	fb103StartQuiescentMode.ipDALICommunication := ipDALICommunication;
	fb103StopQuiescentMode.ipDALICommunication := ipDALICommunication;
	fb253QueryShortCircuit.ipDALICommunication := ipDALICommunication;
	fb253QueryOpenCircuit.ipDALICommunication := ipDALICommunication;
	fb207QueryLoadDecrease.ipDALICommunication := ipDALICommunication;
	fb207QueryLoadIncrease.ipDALICommunication := ipDALICommunication;
	fb253QueryThermalShutDown.ipDALICommunication := ipDALICommunication;
	fb207QueryThermalOverload.ipDALICommunication := ipDALICommunication;
	fb207QueryReferenceMeasurementFailed.ipDALICommunication := ipDALICommunication;
	fb207QueryDimmingCurve.ipDALICommunication := ipDALICommunication;
	fb207QueryFastFadeTime.ipDALICommunication := ipDALICommunication;
	fb102QueryExtendedVersionNumber.ipDALICommunication := ipDALICommunication;
	fb207ReferenceSystemPower.ipDALICommunication := ipDALICommunication;
	fb207SelectDimmingCurve.ipDALICommunication := ipDALICommunication;
	fb207SetFastFadeTime.ipDALICommunication := ipDALICommunication;
	fb207QueryFeatures.ipDALICommunication := ipDALICommunication;
	fb207QueryControlGearType.ipDALICommunication := ipDALICommunication;
{endregion}
{region "Read Status}
5:
{region "Start Qiescent Mode"}
	fb103StartQuiescentMode(bStart := TRUE,
							eAddressType := Tc3_DALI.E_DALIAddressType.Broadcast,
							eCommandPriority := Tc3_DALI.E_DALICommandPriority.Middle);
	IF (NOT fb103StartQuiescentMode.bBusy) THEN
		fb103StartQuiescentMode(bStart:= FALSE);
		nStep := 10;
	END_IF
{endregion}
10:
{region "Query Short Circuit"}
	fb253QueryShortCircuit(	bStart := TRUE,
							nAddress := nAddress,
							eAddressType := Tc3_DALI.E_DALIAddressType.Short,
							eCommandPriority := Tc3_DALI.E_DALICommandPriority.Middle);
	IF (NOT fb253QueryShortCircuit.bBusy) THEN
		fb253QueryShortCircuit(bStart := FALSE);
		sShortCircuit := SEL(fb253QueryShortCircuit.bLightSourceShortCircuit, 'No', 'Yes');
		nStep := 20;
	END_IF
{endregion}
20:
{region "Query Open Circuit"}
	fb253QueryOpenCircuit(	bStart := TRUE,
							nAddress := nAddress,
							eAddressType := Tc3_DALI.E_DALIAddressType.Short,
							eCommandPriority := Tc3_DALI.E_DALICommandPriority.Middle);
	IF (NOT fb253QueryOpenCircuit.bBusy) THEN
		fb253QueryOpenCircuit(bStart := FALSE);
		sOpenCircuit := SEL(fb253QueryOpenCircuit.bLightSourceOpenCircuit, 'No', 'Yes');
		nStep := 30;
	END_IF
{endregion}
30:
{region "Query Load Decrease"}
	fb207QueryLoadDecrease(	bStart := TRUE,
							nAddress := nAddress,
							eAddressType := Tc3_DALI.E_DALIAddressType.Short,
							eCommandPriority := Tc3_DALI.E_DALICommandPriority.Middle);
	IF (NOT fb207QueryLoadDecrease.bBusy) THEN
		fb207QueryLoadDecrease(bStart := FALSE);
		sLoadDecrease := SEL(fb207QueryLoadDecrease.bLoadDecrease, 'No', 'Yes');
		nStep := 40;
	END_IF
{endregion}
40:
{region "Query Load Increase"}
	fb207QueryLoadIncrease(	bStart := TRUE,
							nAddress := nAddress,
							eAddressType := Tc3_DALI.E_DALIAddressType.Short,
							eCommandPriority := Tc3_DALI.E_DALICommandPriority.Middle);
	IF (NOT fb207QueryLoadIncrease.bBusy) THEN
		fb207QueryLoadIncrease(bStart := FALSE);
		sLoadIncrease := SEL(fb207QueryLoadIncrease.bLoadIncrease, 'No', 'Yes');
		nStep := 80;
	END_IF
{endregion}
80:
{region "Query Thermal Shut Down"}
	fb253QueryThermalShutDown(	bStart := TRUE,
								nAddress := nAddress,
								eAddressType := Tc3_DALI.E_DALIAddressType.Short,
								eCommandPriority := Tc3_DALI.E_DALICommandPriority.Middle);
	IF (NOT fb253QueryThermalShutDown.bBusy) THEN
		fb253QueryThermalShutDown(bStart := FALSE);
		sThermalShutDown := SEL(fb253QueryThermalShutDown.bLightSourceThermalShutdown, 'No', 'Yes');
		nStep := 90;
	END_IF
{endregion}
90:
{region "Query Thermal Overload"}
	fb207QueryThermalOverload(	bStart := TRUE,
								nAddress := nAddress,
								eAddressType := Tc3_DALI.E_DALIAddressType.Short,
								eCommandPriority := Tc3_DALI.E_DALICommandPriority.Middle);
	IF (NOT fb207QueryThermalOverload.bBusy) THEN
		fb207QueryThermalOverload(bStart := FALSE);
		sThermalOverload := SEL(fb207QueryThermalOverload.bThermalOverload, 'No', 'Yes');
		nStep := 100;
	END_IF
{endregion}
100:
{region "Query Reference Measurement Failed"}
	fb207QueryReferenceMeasurementFailed(	bStart := TRUE,
											nAddress := nAddress,
											eAddressType := Tc3_DALI.E_DALIAddressType.Short,
											eCommandPriority := Tc3_DALI.E_DALICommandPriority.Middle);
	IF (NOT fb207QueryReferenceMeasurementFailed.bBusy) THEN
		fb207QueryReferenceMeasurementFailed(bStart := FALSE);
		sReferenceMeasurementFailed := SEL(fb207QueryReferenceMeasurementFailed.bReferenceMeasurementFailed, 'No', 'Yes');
		nStep := 110;
	END_IF
{endregion}
110:
{region "Query Dimming Curve"}
	fb207QueryDimmingCurve(	bStart := TRUE,
							nAddress := nAddress,
							eAddressType := Tc3_DALI.E_DALIAddressType.Short,
							eCommandPriority := Tc3_DALI.E_DALICommandPriority.Middle,
							eDimmingCurve => eDimmingCurve);
	IF (NOT fb207QueryDimmingCurve.bBusy) THEN
		fb207QueryDimmingCurve(bStart := FALSE);
		nStep := 120;
	END_IF
{endregion}
120:
{region "Query Fast Fade Time"}
	fb207QueryFastFadeTime(	bStart := TRUE,
							nAddress := nAddress,
							eAddressType := Tc3_DALI.E_DALIAddressType.Short,
							eCommandPriority := Tc3_DALI.E_DALICommandPriority.Middle,
							eFastFadeTime => eFastFadeTime);
	IF (NOT fb207QueryFastFadeTime.bBusy) THEN
		fb207QueryFastFadeTime(bStart := FALSE);
		nStep := 130;
	END_IF
{endregion}
130:
{region "Query Extended Version Number"}
	fb102QueryExtendedVersionNumber(bStart := TRUE,
									nAddress := nAddress,
									eAddressType := Tc3_DALI.E_DALIAddressType.Short,
									eCommandPriority := Tc3_DALI.E_DALICommandPriority.Middle,
									eDeviceType := E_DALIDeviceType.DT06LEDModule,
									nExtendedVersionNumber => nExtendedVersionNumber);
	IF (NOT fb102QueryExtendedVersionNumber.bBusy) THEN
		fb102QueryExtendedVersionNumber(bStart := FALSE);
		nStep := 135;
	END_IF
{endregion}
135:
{region "Stop Qiescent Mode"}
	fb103StopQuiescentMode(	bStart := TRUE,
							eAddressType := Tc3_DALI.E_DALIAddressType.Broadcast,
							eCommandPriority := Tc3_DALI.E_DALICommandPriority.Middle);
	IF (NOT fb103StopQuiescentMode.bBusy) THEN
		fb103StopQuiescentMode(	bStart := FALSE);
		nStep := 0;
	END_IF
{endregion}
{endregion}

{region "Read Parameter"}
200:
{region "Start Qiescent Mode"}
	fb103StartQuiescentMode(bStart := TRUE,
							eAddressType := Tc3_DALI.E_DALIAddressType.Broadcast,
							eCommandPriority := Tc3_DALI.E_DALICommandPriority.Middle);
	IF (NOT fb103StartQuiescentMode.bBusy) THEN
		fb103StartQuiescentMode(bStart:= FALSE);
		nStep := 210;
	END_IF
{endregion}
210:
{region "Query Features"}
	fb207QueryFeatures(	bStart := TRUE,
						nAddress := nAddress,
						eAddressType := Tc3_DALI.E_DALIAddressType.Short,
						eCommandPriority := Tc3_DALI.E_DALICommandPriority.Middle,
						nFeatures => nFeatures);

	IF (NOT fb207QueryFeatures.bBusy) THEN
		fb207QueryFeatures(bStart := FALSE);
		bQueryShortCircuitEnabled := nFeatures.0;
		bQueryIdleTimeDetectionEnabled := nFeatures.1;
		bQueryLoadDecreaseEnabled := nFeatures.2;
		bQueryLoadIncreaseEnabled := nFeatures.3;
		bQueryCurrentProtectionDevicePresent := nFeatures.4;
		bQueryThermalSwitchEnabled := nFeatures.5;
		bQueryReductionOfLuminouFluxRegardingThermalOverloadEnabled := nFeatures.6;
		bPhysicalSelectionSupported := nFeatures.7;
		nStep := 215;
	END_IF
{endregion}
215:
{region "Query control Gear Type"}
	fb207QueryControlGearType(	bStart := TRUE, 
								nAddress := nAddress,
								eAddressType := Tc3_DALI.E_DALIAddressType.Short,
								eCommandPriority := Tc3_DALI.E_DALICommandPriority.Middle,
								nControlGearType => nControlGearType);
	IF (NOT fb207QueryControlGearType.bBusy) THEN
		fb207QueryControlGearType(bStart := FALSE);
		bLEDModule	:= nControlGearType.1;
		nStep := 220;
	END_IF
{endregion}
220:
{region "Stop Qiescent Mode"}
	fb103StopQuiescentMode(	bStart := TRUE,
							eAddressType := Tc3_DALI.E_DALIAddressType.Broadcast,
							eCommandPriority := Tc3_DALI.E_DALICommandPriority.Middle);
	IF (NOT fb103StopQuiescentMode.bBusy) THEN
		fb103StopQuiescentMode(	bStart := FALSE);
		nStep := 0;
	END_IF
{endregion}
{endregion}

{region "Write"}
1000:
{region "Reference System Power"}
	fb207ReferenceSystemPower(	bStart := TRUE,
								nAddress := nAddress,
								eAddressType := Tc3_DALI.E_DALIAddressType.Short,
								eCommandPriority := Tc3_DALI.E_DALICommandPriority.Middle);
	IF (NOT fb207ReferenceSystemPower.bBusy) THEN
		fb207ReferenceSystemPower(bStart := FALSE);
		nStep := 0;
	END_IF
{endregion}
1030:
{region "Select Dimming Curve"}
	fb207SelectDimmingCurve(bStart := TRUE,
							nAddress := nAddress,
							eAddressType := Tc3_DALI.E_DALIAddressType.Short,
							eCommandPriority := Tc3_DALI.E_DALICommandPriority.Middle,
							eDimmingCurve := eDimmingCurve);
	IF (NOT fb207SelectDimmingCurve.bBusy) THEN
		fb207SelectDimmingCurve(bStart := FALSE);
		nStep := 1040;
	END_IF
{endregion}
1040:
{region "Set Fast Fade Time"}
	fb207SetFastFadeTime(bStart := TRUE,
						nAddress := nAddress,
						eAddressType := Tc3_DALI.E_DALIAddressType.Short,
						eCommandPriority := Tc3_DALI.E_DALICommandPriority.Middle,
						eFastFadeTime := eFastFadeTime);
	IF (NOT fb207SetFastFadeTime.bBusy) THEN
		fb207SetFastFadeTime(bStart := FALSE);
		nStep := 0;
	END_IF
{endregion}
{endregion}
END_CASE

END_FUNCTION_BLOCK

// ---- POUs/EnOcean/P_EnOcean.TcPOU
PROGRAM P_EnOcean
VAR
	fbKL6581			: FB_KL6581;
	stKL6581_in  AT %I* : KL6581_INPUT;
	stKL6581_out AT %Q*	: KL6581_OUTPUT;
	stKL6581			: STR_KL6581;
	bInitCom			: BOOL := TRUE;
	
	arrEnOcean_Search	: ARRAY [1..8] OF FB_EnOcean_Search;
	nSearchIdx			: BYTE;
	bSerach				: BOOL;
	arrDevices			: ARRAY [1..8] OF INT;
	arrID					: ARRAY [1..8, 0..255] OF DWORD;

	//Trykknapper på gange
	fbGang_1_216_Tryk_Pendler    							: FB_Rec_RPS_Switch;	
	
	//Trykknapper i rum
	fbRum_1_213_Tryk_Indgang								: FB_Rec_RPS_Switch;
	fbRum_1_213_Tryk_Ekstra								: FB_Rec_RPS_Switch;
	
	fbRum_1_215_Tryk											: FB_Rec_RPS_Switch;
	fbRum_1_217_Tryk											: FB_Rec_RPS_Switch;
	fbRum_1_218_Tryk											: FB_Rec_RPS_Switch;
	fbRum_1_219_Tryk											: FB_Rec_RPS_Switch;
	fbRum_1_220_Tryk											: FB_Rec_RPS_Switch;
	fbRum_1_222_Tryk											: FB_Rec_RPS_Switch;
	fbRum_1_223_Tryk											: FB_Rec_RPS_Switch;
	
	fbRum_6_223_Tryk											: FB_Rec_RPS_Switch;
	fbRum_6_224_Tryk											: FB_Rec_RPS_Switch;
	fbRum_6_225_Tryk											: FB_Rec_RPS_Switch;
	fbRum_6_226A_Tryk										: FB_Rec_RPS_Switch;
	
	fbRum_6_226B_Tryk_Indgang							: FB_Rec_RPS_Switch;
	fbRum_6_226B_Tryk_Pendler							: FB_Rec_RPS_Switch;
	
	fbRum_6_227_Tryk											: FB_Rec_RPS_Switch;
	fbRum_6_228_Tryk											: FB_Rec_RPS_Switch;
	fbRum_6_229_Tryk											: FB_Rec_RPS_Switch;
	fbRum_6_230_Tryk											: FB_Rec_RPS_Switch;
	fbRum_6_231_Tryk											: FB_Rec_RPS_Switch;
	fbRum_6_233_Tryk											: FB_Rec_RPS_Switch;
	
	fbRum_6_235_Tryk_Indgang								: FB_Rec_RPS_Switch;
	fbRum_6_235_Tryk_Ekstra								: FB_Rec_RPS_Switch;
	
	
END_VAR

VAR CONSTANT
	byNode_1: BYTE := 1;
	byNode_2: BYTE := 2;
	byNode_3: BYTE := 3;
	byNode_4: BYTE := 4;
	byNode_5: BYTE := 5;
	byNode_6: BYTE := 6;
	byNode_7: BYTE := 7;
	byNode_8: BYTE := 8;
END_VAR


(* Kommunikation mit der KL6581. *)
(* Communication with the KL6581. *)
fbKL6581(
	bInit			:= bInitCom,
	nIdx			:= 2,
	stKL6581_in		:= stKL6581_In,
	stKL6581_out	:= stKL6581_Out,
	bReady			=> ,
	bBusy			=> ,
	bError			=> ,
	iErrorID		=> ,
	str_KL6581		=> stKL6581);
	
GVL_AHDataModbus.EnOceanError	:= TO_UINT(fbKL6581.iErrorID);

(* Warten bis der Kommunikationsbaustein initialisiert wurde.*)
(* Wait until the communication function block has been initialized. *)
IF (NOT fbKL6581.bReady) THEN
	RETURN;
END_IF

FOR nSearchIdx:= 1 TO 8 DO
	arrEnOcean_Search[nSearchIdx](
		bStart:= TRUE, 
		str_KL6581:= stKL6581 , 
		byNode:= nSearchIdx, 
		bReceive=> , 
		iDevices=>arrDevices[nSearchIdx] , 
		ar_ID=> );
		
		MEMCPY(ADR(arrID[nSearchIdx,0]), ADR(arrEnOcean_Search[nSearchIdx].ar_ID), SIZEOF(arrEnOcean_Search[nSearchIdx].ar_ID)); 
END_FOR

//Gange
A_Gang_1_216();

//Rum
A_Rum_1_213();
A_Rum_1_215();
A_Rum_1_217();
A_Rum_1_218();
A_Rum_1_219();
A_Rum_1_220();
A_Rum_1_222();
A_Rum_1_223();

A_Rum_6_223();
A_Rum_6_224();
A_Rum_6_225();
A_Rum_6_226A();
A_Rum_6_226B();
A_Rum_6_227();
A_Rum_6_228();
A_Rum_6_229();
A_Rum_6_230();
A_Rum_6_231();
A_Rum_6_233();
A_Rum_6_235();

ACTION A_Gang_1_216:
fbGang_1_216_Tryk_Pendler(
	str_KL6581:=stKL6581 , 
	byNode:=byNode_2, 
	dw_ID:= 16#002AC914, 
	str_EnOceanSwitch=> GVL_EnOcean.strEnOceanSwitch_Gang_1_216_Pendler, 
	by_Node=> , 
	bReceive=> );
END_ACTION

ACTION A_Rum_1_213:
fbRum_1_213_Tryk_Indgang(
	str_KL6581:=stKL6581 , 
	byNode:=byNode_2, 
	dw_ID:= 16#0029AD59, 
	str_EnOceanSwitch=> GVL_EnOcean.strEnOceanSwitch_Rum_1_213_Indgang, 
	by_Node=> , 
	bReceive=> );
	
	fbRum_1_213_Tryk_Ekstra(
	str_KL6581:=stKL6581 , 
	byNode:=byNode_2, 
	dw_ID:= 16#0029AD60, 
	str_EnOceanSwitch=> GVL_EnOcean.strEnOceanSwitch_Rum_1_213_Ekstra, 
	by_Node=> , 
	bReceive=> );
END_ACTION

ACTION A_Rum_1_215:
fbRum_1_215_Tryk(
	str_KL6581:=stKL6581 , 
	byNode:=byNode_2, 
	dw_ID:= 16#0029AD91, 
	str_EnOceanSwitch=> GVL_EnOcean.strEnOceanSwitch_Rum_1_215, 
	by_Node=> , 
	bReceive=> );
END_ACTION

ACTION A_Rum_1_217:
fbRum_1_217_Tryk(
	str_KL6581:=stKL6581 , 
	byNode:=byNode_2, 
	dw_ID:= 16#0029AD6B, 
	str_EnOceanSwitch=> GVL_EnOcean.strEnOceanSwitch_Rum_1_217, 
	by_Node=> , 
	bReceive=> );
END_ACTION

ACTION A_Rum_1_218:
fbRum_1_218_Tryk(
	str_KL6581:=stKL6581 , 
	byNode:=byNode_2, 
	dw_ID:= 16#0029AAFF, 
	str_EnOceanSwitch=> GVL_EnOcean.strEnOceanSwitch_Rum_1_218, 
	by_Node=> , 
	bReceive=> );
END_ACTION

ACTION A_Rum_1_219:
fbRum_1_219_Tryk(
	str_KL6581:=stKL6581 , 
	byNode:=byNode_2, 
	dw_ID:= 16#0029AD67, 
	str_EnOceanSwitch=> GVL_EnOcean.strEnOceanSwitch_Rum_1_219, 
	by_Node=> , 
	bReceive=> );
END_ACTION

ACTION A_Rum_1_220:
fbRum_1_220_Tryk(
	str_KL6581:=stKL6581 , 
	byNode:=byNode_2, 
	dw_ID:= 16#0029AD83, 
	str_EnOceanSwitch=> GVL_EnOcean.strEnOceanSwitch_Rum_1_220, 
	by_Node=> , 
	bReceive=> );
END_ACTION

ACTION A_Rum_1_222:
fbRum_1_222_Tryk(
	str_KL6581:=stKL6581 , 
	byNode:=byNode_2, 
	dw_ID:= 16#0029AB84, 
	str_EnOceanSwitch=> GVL_EnOcean.strEnOceanSwitch_Rum_1_222, 
	by_Node=> , 
	bReceive=> );
END_ACTION

ACTION A_Rum_1_223:
fbRum_1_223_Tryk(
	str_KL6581:=stKL6581 , 
	byNode:=byNode_2, 
	dw_ID:=16#0029AD46, 
	str_EnOceanSwitch=> GVL_EnOcean.strEnOceanSwitch_Rum_1_223, 
	by_Node=> , 
	bReceive=> );
END_ACTION

ACTION A_Rum_6_223:
fbRum_6_223_Tryk(
	str_KL6581:=stKL6581 , 
	byNode:=byNode_2, 
	dw_ID:= 16#0029AAF4, 
	str_EnOceanSwitch=> GVL_EnOcean.strEnOceanSwitch_Rum_6_223, 
	by_Node=> , 
	bReceive=> );
END_ACTION

ACTION A_Rum_6_224:
fbRum_6_224_Tryk(
	str_KL6581:=stKL6581 , 
	byNode:=byNode_2, 
	dw_ID:= 16#0029AD78, 
	str_EnOceanSwitch=> GVL_EnOcean.strEnOceanSwitch_Rum_6_224, 
	by_Node=> , 
	bReceive=> );
END_ACTION

ACTION A_Rum_6_225:
fbRum_6_225_Tryk(
	str_KL6581:=stKL6581 , 
	byNode:=byNode_2, 
	dw_ID:= 16#0029AAED, 
	str_EnOceanSwitch=> GVL_EnOcean.strEnOceanSwitch_Rum_6_225, 
	by_Node=> , 
	bReceive=> );
END_ACTION

ACTION A_Rum_6_226A:
fbRum_6_226A_Tryk(
	str_KL6581:=stKL6581 , 
	byNode:=byNode_2, 
	dw_ID:= 16#0029AD5C, 
	str_EnOceanSwitch=> GVL_EnOcean.strEnOceanSwitch_Rum_6_226A, 
	by_Node=> , 
	bReceive=> );
END_ACTION

ACTION A_Rum_6_226B:
fbRum_6_226B_Tryk_Indgang(
	str_KL6581:=stKL6581 , 
	byNode:=byNode_2, 
	dw_ID:= 16#0029AD81, 
	str_EnOceanSwitch=> GVL_EnOcean.strEnOceanSwitch_Rum_6_226B_Indgang, 
	by_Node=> , 
	bReceive=> );
	
	fbRum_6_226B_Tryk_Pendler(
	str_KL6581:=stKL6581 , 
	byNode:=byNode_2, 
	dw_ID:= 16#FEE507E2, 
	str_EnOceanSwitch=> GVL_EnOcean.strEnOceanSwitch_Rum_6_226B_Pendler, 
	by_Node=> , 
	bReceive=> );
END_ACTION

ACTION A_Rum_6_227:
fbRum_6_227_Tryk(
	str_KL6581:=stKL6581 , 
	byNode:=byNode_2, 
	dw_ID:= 16#0029AAF7, 
	str_EnOceanSwitch=> GVL_EnOcean.strEnOceanSwitch_Rum_6_227, 
	by_Node=> , 
	bReceive=> );
END_ACTION

ACTION A_Rum_6_228:
fbRum_6_228_Tryk(
	str_KL6581:=stKL6581 , 
	byNode:=byNode_2, 
	dw_ID:= 16#0029AD7C, 
	str_EnOceanSwitch=> GVL_EnOcean.strEnOceanSwitch_Rum_6_228, 
	by_Node=> , 
	bReceive=> );
END_ACTION

ACTION A_Rum_6_229:
fbRum_6_229_Tryk(
	str_KL6581:=stKL6581 , 
	byNode:=byNode_2, 
	dw_ID:= 16#0029AD85, 
	str_EnOceanSwitch=> GVL_EnOcean.strEnOceanSwitch_Rum_6_229, 
	by_Node=> , 
	bReceive=> );
END_ACTION

ACTION A_Rum_6_230:
fbRum_6_230_Tryk(
	str_KL6581:=stKL6581 , 
	byNode:=byNode_2, 
	dw_ID:= 16#0029AAFA, 
	str_EnOceanSwitch=> GVL_EnOcean.strEnOceanSwitch_Rum_6_230, 
	by_Node=> , 
	bReceive=> );
END_ACTION

ACTION A_Rum_6_231:
fbRum_6_231_Tryk(
	str_KL6581:=stKL6581 , 
	byNode:=byNode_2, 
	dw_ID:= 16#0029AD6A, 
	str_EnOceanSwitch=> GVL_EnOcean.strEnOceanSwitch_Rum_6_231, 
	by_Node=> , 
	bReceive=> );
END_ACTION

ACTION A_Rum_6_233:
fbRum_6_233_Tryk(
	str_KL6581:=stKL6581 , 
	byNode:=byNode_2, 
	dw_ID:= 16#0029AD5F, 
	str_EnOceanSwitch=> GVL_EnOcean.strEnOceanSwitch_Rum_6_233, 
	by_Node=> , 
	bReceive=> );
END_ACTION

ACTION A_Rum_6_235:
fbRum_6_235_Tryk_Indgang(
	str_KL6581:=stKL6581 , 
	byNode:=byNode_2, 
	dw_ID:= 16#0029AD72, 
	str_EnOceanSwitch=> GVL_EnOcean.strEnOceanSwitch_Rum_6_235_Indgang, 
	by_Node=> , 
	bReceive=> );
	
	fbRum_6_235_Tryk_Ekstra(
	str_KL6581:=stKL6581 , 
	byNode:=byNode_2, 
	dw_ID:= 16#0029AD5D, 
	str_EnOceanSwitch=> GVL_EnOcean.strEnOceanSwitch_Rum_6_235_Ekstra, 
	by_Node=> , 
	bReceive=> );
END_ACTION

END_PROGRAM

// ---- POUs/MAIN.TcPOU
PROGRAM MAIN
VAR
	nAlive: INT;
	breset: BOOL;
	nDemoVariable : INT;
	nCX8200_State	AT %I*	: UINT;
END_VAR

VAR PERSISTENT
	nDemoVar_Persist: INT;
END_VAR

nAlive:= nAlive + 1;
GVL_AHDataModbus.nCX8200_State_MB := nCX8200_State;

//Håndterer vedvarende data
	P_SystemDK.M_nCyclic(bReset := breset );
//Håndterer DALI-diagnostik (run once)
	P_DALI_DIAG();
//Håndterer adressering		
	DALI_Commissioning();
//Håndterer energirapportering
	P_DALI_Energy_Line();
//Håndterer moodbus-kommunikation (kun PLC-oversigt)
	P_AHModbusComm();

//Håndterer individuel lyskontrol i lokaler
	//Gange
	P_Gang_1_212A();
	P_Gang_1_216();
	P_Gang_6_210();
	
	//Rum
	P_Rum_1_213();
	P_Rum_1_215();
	P_Rum_1_217();
	P_Rum_1_218();
	P_Rum_1_219();
	P_Rum_1_220();
	P_Rum_1_222();
	P_Rum_1_223();
	
	P_Rum_6_223();
	P_Rum_6_224();
	P_Rum_6_225();
	P_Rum_6_226A();
	P_rum_6_226B();
	P_Rum_6_227();
	P_Rum_6_228();
	P_Rum_6_229();
	P_Rum_6_230();
	P_Rum_6_231();
	P_Rum_6_233();
	P_Rum_6_235();

	


	//Trapper
	//P_Trappe();
	
//Testprogrammer
	//P_DALI_Energy_Firmware_Test();

END_PROGRAM

// ---- POUs/Alle_Rum/Gange/Gang_1_212A/Visualization_4_307_1_1_1_1.TcVIS
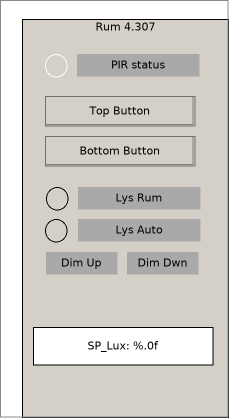
VISUALIZATION Visualization_4_307_1_1_1_1  // 229x418
    RoundedRectangle (22,19 207x399), "Rum 4.307"
    Rectangle (33,327 180x38), "SP_Lux: %.0f", text variable: P_Rum_4_307.fbLys.fbLightCtrl.fLuxZone1
    Button (45,96 150x30), "Top Button"
        tap P_Rum_4_307.bTopButtonZone1_Visu
    Button (45,136 150x30), "Bottom Button"
        tap P_Rum_4_307.bBottomButtonZone1_Visu
    Ellipse (46,187 22x23), colour toggle: P_Rum_4_307.fbLys.fbLightCtrl.bOnZone1
    Rectangle (78,187 122x22), "Lys Rum"
    Rectangle (46,252 71x22), "Dim Up", colour toggle: P_Rum_4_307.fbLys.fbLightCtrl.bDimUp
    Rectangle (127,252 71x22), "Dim Dwn", colour toggle: P_Rum_4_307.fbLys.fbLightCtrl.bDimDwn
    Ellipse (45,219 22x23), colour toggle: P_Rum_4_307.fbLys.fbLightCtrl.bAutoZone1
    Rectangle (78,219 122x22), "Lys Auto"
    Ellipse (45,54 22x23), colour toggle: P_Rum_4_307.fbLys.fbLightCtrl.bPIR
    Rectangle (77,54 122x22), "PIR status"
END_VISUALIZATION

// ---- POUs/Alle_Rum/Gange/Gang_1_216/Visualization_4_308_1_2_1.TcVIS
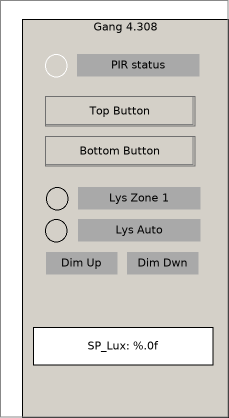
VISUALIZATION Visualization_4_308_1_2_1  // 229x418
    RoundedRectangle (22,19 207x399), "Gang 4.308"
    Rectangle (33,327 180x38), "SP_Lux: %.0f", text variable: P_Gang_4_308.arrfbLysGruppe[1].fbLightCtrl.fLuxZone1
    Button (45,96 150x30), "Top Button"
        tap P_Gang_4_308.bButtonZone1_Visu
    Button (45,136 150x30), "Bottom Button"
        tap P_Gang_4_308.bBottomButtonZone1_Visu
    Ellipse (46,187 22x23), colour toggle: P_Gang_4_308.fbLys.fbLightCtrl.bOnZone1
    Rectangle (78,187 122x22), "Lys Zone 1"
    Rectangle (46,252 71x22), "Dim Up", colour toggle: P_Gang_4_308.arrfbLysGruppe[1].fbLightCtrl.bDimUp
    Rectangle (127,252 71x22), "Dim Dwn", colour toggle: P_Gang_4_308.arrfbLysGruppe[1].fbLightCtrl.bDimDwn
    Ellipse (45,219 22x23), colour toggle: P_Gang_4_308.arrfbLysGruppe[1].fbLightCtrl.bAutoZone1
    Rectangle (78,219 122x22), "Lys Auto"
    Ellipse (45,54 22x23), colour toggle: P_Gang_4_308.arrfbLysGruppe[1].fbLightCtrl.bPIR
    Rectangle (77,54 122x22), "PIR status"
END_VISUALIZATION

// ---- POUs/Alle_Rum/Gange/Gang_6_210/Visualization_4_308_1_2_1_1.TcVIS
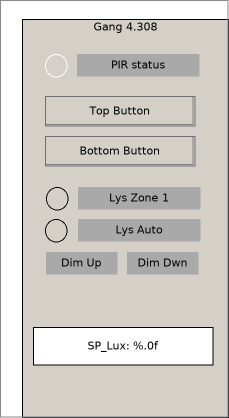
VISUALIZATION Visualization_4_308_1_2_1_1  // 229x418
    RoundedRectangle (22,19 207x399), "Gang 4.308"
    Rectangle (33,327 180x38), "SP_Lux: %.0f", text variable: P_Gang_4_308.arrfbLysGruppe[1].fbLightCtrl.fLuxZone1
    Button (45,96 150x30), "Top Button"
        tap P_Gang_4_308.bButtonZone1_Visu
    Button (45,136 150x30), "Bottom Button"
        tap P_Gang_4_308.bBottomButtonZone1_Visu
    Ellipse (46,187 22x23), colour toggle: P_Gang_4_308.fbLys.fbLightCtrl.bOnZone1
    Rectangle (78,187 122x22), "Lys Zone 1"
    Rectangle (46,252 71x22), "Dim Up", colour toggle: P_Gang_4_308.arrfbLysGruppe[1].fbLightCtrl.bDimUp
    Rectangle (127,252 71x22), "Dim Dwn", colour toggle: P_Gang_4_308.arrfbLysGruppe[1].fbLightCtrl.bDimDwn
    Ellipse (45,219 22x23), colour toggle: P_Gang_4_308.arrfbLysGruppe[1].fbLightCtrl.bAutoZone1
    Rectangle (78,219 122x22), "Lys Auto"
    Ellipse (45,54 22x23), colour toggle: P_Gang_4_308.arrfbLysGruppe[1].fbLightCtrl.bPIR
    Rectangle (77,54 122x22), "PIR status"
END_VISUALIZATION

// ---- POUs/Alle_Rum/Rum_Med_DALI_Pir/Rum_1_213/Visualization_5_356_2_1_1_1.TcVIS
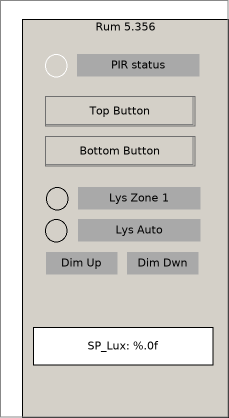
VISUALIZATION Visualization_5_356_2_1_1_1  // 229x418
    RoundedRectangle (22,19 207x399), "Rum 5.356"
    Rectangle (33,327 180x38), "SP_Lux: %.0f", text variable: P_Rum_5_356.arrfbLysGruppe[1].fbLightCtrl.fLuxZone1
    Button (45,96 150x30), "Top Button"
        tap P_Rum_5_356.bTopButtonZone1_Visu
    Button (45,136 150x30), "Bottom Button"
        tap P_Rum_5_356.bBottomButtonZone1_Visu
    Ellipse (46,187 22x23), colour toggle: P_Rum_5_356.arrfbLysGruppe[1].fbLightCtrl.bOnZone1
    Rectangle (78,187 122x22), "Lys Zone 1"
    Rectangle (46,252 71x22), "Dim Up", colour toggle: P_Rum_5_356.arrfbLysGruppe[1].fbLightCtrl.bDimUp
    Rectangle (127,252 71x22), "Dim Dwn", colour toggle: P_Rum_5_356.arrfbLysGruppe[1].fbLightCtrl.bDimDwn
    Ellipse (45,219 22x23), colour toggle: P_Rum_5_356.arrfbLysGruppe[1].fbLightCtrl.bAutoZone1
    Rectangle (78,219 122x22), "Lys Auto"
    Ellipse (45,54 22x23), colour toggle: P_Gang_5_356.arrfbLysGruppe[1].fbLightCtrl.bPIR
    Rectangle (77,54 122x22), "PIR status"
END_VISUALIZATION

// ---- POUs/Alle_Rum/Rum_Med_DALI_Pir/Rum_6_235/Visualization_5_356_2_1_1_1_1.TcVIS
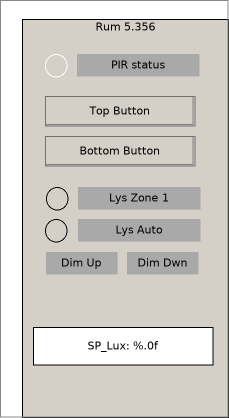
VISUALIZATION Visualization_5_356_2_1_1_1_1  // 229x418
    RoundedRectangle (22,19 207x399), "Rum 5.356"
    Rectangle (33,327 180x38), "SP_Lux: %.0f", text variable: P_Rum_5_356.arrfbLysGruppe[1].fbLightCtrl.fLuxZone1
    Button (45,96 150x30), "Top Button"
        tap P_Rum_5_356.bTopButtonZone1_Visu
    Button (45,136 150x30), "Bottom Button"
        tap P_Rum_5_356.bBottomButtonZone1_Visu
    Ellipse (46,187 22x23), colour toggle: P_Rum_5_356.arrfbLysGruppe[1].fbLightCtrl.bOnZone1
    Rectangle (78,187 122x22), "Lys Zone 1"
    Rectangle (46,252 71x22), "Dim Up", colour toggle: P_Rum_5_356.arrfbLysGruppe[1].fbLightCtrl.bDimUp
    Rectangle (127,252 71x22), "Dim Dwn", colour toggle: P_Rum_5_356.arrfbLysGruppe[1].fbLightCtrl.bDimDwn
    Ellipse (45,219 22x23), colour toggle: P_Rum_5_356.arrfbLysGruppe[1].fbLightCtrl.bAutoZone1
    Rectangle (78,219 122x22), "Lys Auto"
    Ellipse (45,54 22x23), colour toggle: P_Gang_5_356.arrfbLysGruppe[1].fbLightCtrl.bPIR
    Rectangle (77,54 122x22), "PIR status"
END_VISUALIZATION

// ---- POUs/Alle_Rum/Rum_Med_DALI_Pir/Rum_1_215/Visualization_4_307_1_1_3_1_1_1.TcVIS
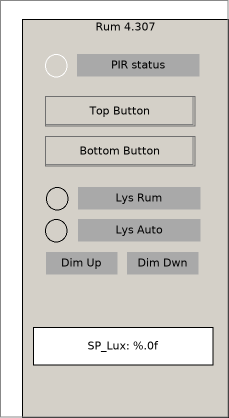
VISUALIZATION Visualization_4_307_1_1_3_1_1_1  // 229x418
    RoundedRectangle (22,19 207x399), "Rum 4.307"
    Rectangle (33,327 180x38), "SP_Lux: %.0f", text variable: P_Rum_4_307.fbLys.fbLightCtrl.fLuxZone1
    Button (45,96 150x30), "Top Button"
        tap P_Rum_4_307.bTopButtonZone1_Visu
    Button (45,136 150x30), "Bottom Button"
        tap P_Rum_4_307.bBottomButtonZone1_Visu
    Ellipse (46,187 22x23), colour toggle: P_Rum_4_307.fbLys.fbLightCtrl.bOnZone1
    Rectangle (78,187 122x22), "Lys Rum"
    Rectangle (46,252 71x22), "Dim Up", colour toggle: P_Rum_4_307.fbLys.fbLightCtrl.bDimUp
    Rectangle (127,252 71x22), "Dim Dwn", colour toggle: P_Rum_4_307.fbLys.fbLightCtrl.bDimDwn
    Ellipse (45,219 22x23), colour toggle: P_Rum_4_307.fbLys.fbLightCtrl.bAutoZone1
    Rectangle (78,219 122x22), "Lys Auto"
    Ellipse (45,54 22x23), colour toggle: P_Rum_4_307.fbLys.fbLightCtrl.bPIR
    Rectangle (77,54 122x22), "PIR status"
END_VISUALIZATION

// ---- POUs/Alle_Rum/Rum_Med_DALI_Pir/Rum_1_217/Visualization_5_356_2_1_1_2.TcVIS
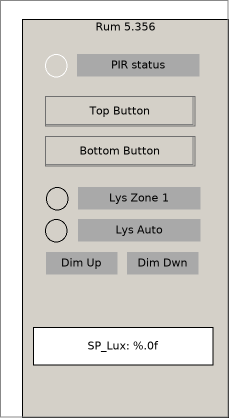
VISUALIZATION Visualization_5_356_2_1_1_2  // 229x418
    RoundedRectangle (22,19 207x399), "Rum 5.356"
    Rectangle (33,327 180x38), "SP_Lux: %.0f", text variable: P_Rum_5_356.arrfbLysGruppe[1].fbLightCtrl.fLuxZone1
    Button (45,96 150x30), "Top Button"
        tap P_Rum_5_356.bTopButtonZone1_Visu
    Button (45,136 150x30), "Bottom Button"
        tap P_Rum_5_356.bBottomButtonZone1_Visu
    Ellipse (46,187 22x23), colour toggle: P_Rum_5_356.arrfbLysGruppe[1].fbLightCtrl.bOnZone1
    Rectangle (78,187 122x22), "Lys Zone 1"
    Rectangle (46,252 71x22), "Dim Up", colour toggle: P_Rum_5_356.arrfbLysGruppe[1].fbLightCtrl.bDimUp
    Rectangle (127,252 71x22), "Dim Dwn", colour toggle: P_Rum_5_356.arrfbLysGruppe[1].fbLightCtrl.bDimDwn
    Ellipse (45,219 22x23), colour toggle: P_Rum_5_356.arrfbLysGruppe[1].fbLightCtrl.bAutoZone1
    Rectangle (78,219 122x22), "Lys Auto"
    Ellipse (45,54 22x23), colour toggle: P_Gang_5_356.arrfbLysGruppe[1].fbLightCtrl.bPIR
    Rectangle (77,54 122x22), "PIR status"
END_VISUALIZATION

// ---- POUs/Alle_Rum/Rum_Med_DALI_Pir/Rum_1_219/Visualization_5_356_2_1_1_3.TcVIS
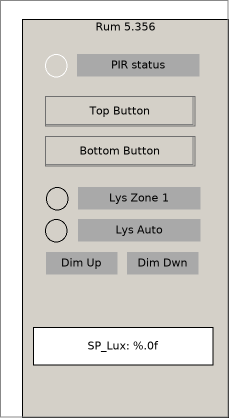
VISUALIZATION Visualization_5_356_2_1_1_3  // 229x418
    RoundedRectangle (22,19 207x399), "Rum 5.356"
    Rectangle (33,327 180x38), "SP_Lux: %.0f", text variable: P_Rum_5_356.arrfbLysGruppe[1].fbLightCtrl.fLuxZone1
    Button (45,96 150x30), "Top Button"
        tap P_Rum_5_356.bTopButtonZone1_Visu
    Button (45,136 150x30), "Bottom Button"
        tap P_Rum_5_356.bBottomButtonZone1_Visu
    Ellipse (46,187 22x23), colour toggle: P_Rum_5_356.arrfbLysGruppe[1].fbLightCtrl.bOnZone1
    Rectangle (78,187 122x22), "Lys Zone 1"
    Rectangle (46,252 71x22), "Dim Up", colour toggle: P_Rum_5_356.arrfbLysGruppe[1].fbLightCtrl.bDimUp
    Rectangle (127,252 71x22), "Dim Dwn", colour toggle: P_Rum_5_356.arrfbLysGruppe[1].fbLightCtrl.bDimDwn
    Ellipse (45,219 22x23), colour toggle: P_Rum_5_356.arrfbLysGruppe[1].fbLightCtrl.bAutoZone1
    Rectangle (78,219 122x22), "Lys Auto"
    Ellipse (45,54 22x23), colour toggle: P_Gang_5_356.arrfbLysGruppe[1].fbLightCtrl.bPIR
    Rectangle (77,54 122x22), "PIR status"
END_VISUALIZATION

// ---- POUs/Alle_Rum/Rum_Med_DALI_Pir/Rum_6_226B/Visualization_5_356_2_1_1_3_1.TcVIS
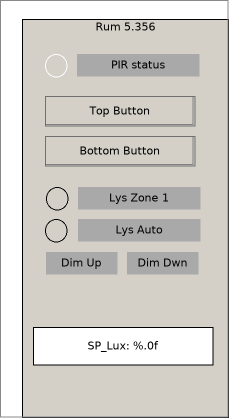
VISUALIZATION Visualization_5_356_2_1_1_3_1  // 229x418
    RoundedRectangle (22,19 207x399), "Rum 5.356"
    Rectangle (33,327 180x38), "SP_Lux: %.0f", text variable: P_Rum_5_356.arrfbLysGruppe[1].fbLightCtrl.fLuxZone1
    Button (45,96 150x30), "Top Button"
        tap P_Rum_5_356.bTopButtonZone1_Visu
    Button (45,136 150x30), "Bottom Button"
        tap P_Rum_5_356.bBottomButtonZone1_Visu
    Ellipse (46,187 22x23), colour toggle: P_Rum_5_356.arrfbLysGruppe[1].fbLightCtrl.bOnZone1
    Rectangle (78,187 122x22), "Lys Zone 1"
    Rectangle (46,252 71x22), "Dim Up", colour toggle: P_Rum_5_356.arrfbLysGruppe[1].fbLightCtrl.bDimUp
    Rectangle (127,252 71x22), "Dim Dwn", colour toggle: P_Rum_5_356.arrfbLysGruppe[1].fbLightCtrl.bDimDwn
    Ellipse (45,219 22x23), colour toggle: P_Rum_5_356.arrfbLysGruppe[1].fbLightCtrl.bAutoZone1
    Rectangle (78,219 122x22), "Lys Auto"
    Ellipse (45,54 22x23), colour toggle: P_Gang_5_356.arrfbLysGruppe[1].fbLightCtrl.bPIR
    Rectangle (77,54 122x22), "PIR status"
END_VISUALIZATION

// ---- POUs/Alle_Rum/Rum_Med_DALI_Pir/Rum_1_220/Visualization_5_356_2_1_1_4.TcVIS
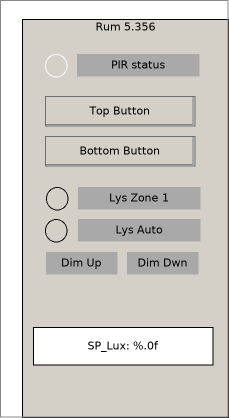
VISUALIZATION Visualization_5_356_2_1_1_4  // 229x418
    RoundedRectangle (22,19 207x399), "Rum 5.356"
    Rectangle (33,327 180x38), "SP_Lux: %.0f", text variable: P_Rum_5_356.arrfbLysGruppe[1].fbLightCtrl.fLuxZone1
    Button (45,96 150x30), "Top Button"
        tap P_Rum_5_356.bTopButtonZone1_Visu
    Button (45,136 150x30), "Bottom Button"
        tap P_Rum_5_356.bBottomButtonZone1_Visu
    Ellipse (46,187 22x23), colour toggle: P_Rum_5_356.arrfbLysGruppe[1].fbLightCtrl.bOnZone1
    Rectangle (78,187 122x22), "Lys Zone 1"
    Rectangle (46,252 71x22), "Dim Up", colour toggle: P_Rum_5_356.arrfbLysGruppe[1].fbLightCtrl.bDimUp
    Rectangle (127,252 71x22), "Dim Dwn", colour toggle: P_Rum_5_356.arrfbLysGruppe[1].fbLightCtrl.bDimDwn
    Ellipse (45,219 22x23), colour toggle: P_Rum_5_356.arrfbLysGruppe[1].fbLightCtrl.bAutoZone1
    Rectangle (78,219 122x22), "Lys Auto"
    Ellipse (45,54 22x23), colour toggle: P_Gang_5_356.arrfbLysGruppe[1].fbLightCtrl.bPIR
    Rectangle (77,54 122x22), "PIR status"
END_VISUALIZATION

// ---- POUs/Alle_Rum/Rum_Med_DALI_Pir/Rum_1_222/Visualization_5_356_2_1_1_5.TcVIS
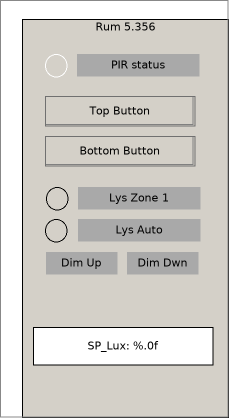
VISUALIZATION Visualization_5_356_2_1_1_5  // 229x418
    RoundedRectangle (22,19 207x399), "Rum 5.356"
    Rectangle (33,327 180x38), "SP_Lux: %.0f", text variable: P_Rum_5_356.arrfbLysGruppe[1].fbLightCtrl.fLuxZone1
    Button (45,96 150x30), "Top Button"
        tap P_Rum_5_356.bTopButtonZone1_Visu
    Button (45,136 150x30), "Bottom Button"
        tap P_Rum_5_356.bBottomButtonZone1_Visu
    Ellipse (46,187 22x23), colour toggle: P_Rum_5_356.arrfbLysGruppe[1].fbLightCtrl.bOnZone1
    Rectangle (78,187 122x22), "Lys Zone 1"
    Rectangle (46,252 71x22), "Dim Up", colour toggle: P_Rum_5_356.arrfbLysGruppe[1].fbLightCtrl.bDimUp
    Rectangle (127,252 71x22), "Dim Dwn", colour toggle: P_Rum_5_356.arrfbLysGruppe[1].fbLightCtrl.bDimDwn
    Ellipse (45,219 22x23), colour toggle: P_Rum_5_356.arrfbLysGruppe[1].fbLightCtrl.bAutoZone1
    Rectangle (78,219 122x22), "Lys Auto"
    Ellipse (45,54 22x23), colour toggle: P_Gang_5_356.arrfbLysGruppe[1].fbLightCtrl.bPIR
    Rectangle (77,54 122x22), "PIR status"
END_VISUALIZATION

// ---- POUs/Alle_Rum/Rum_Med_DALI_Pir/Rum_1_223/Visualization_5_356_2_1_1_6.TcVIS
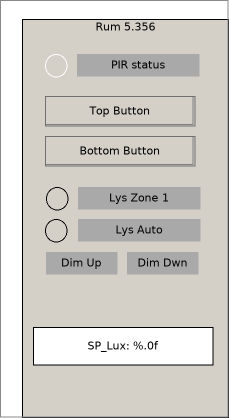
VISUALIZATION Visualization_5_356_2_1_1_6  // 229x418
    RoundedRectangle (22,19 207x399), "Rum 5.356"
    Rectangle (33,327 180x38), "SP_Lux: %.0f", text variable: P_Rum_5_356.arrfbLysGruppe[1].fbLightCtrl.fLuxZone1
    Button (45,96 150x30), "Top Button"
        tap P_Rum_5_356.bTopButtonZone1_Visu
    Button (45,136 150x30), "Bottom Button"
        tap P_Rum_5_356.bBottomButtonZone1_Visu
    Ellipse (46,187 22x23), colour toggle: P_Rum_5_356.arrfbLysGruppe[1].fbLightCtrl.bOnZone1
    Rectangle (78,187 122x22), "Lys Zone 1"
    Rectangle (46,252 71x22), "Dim Up", colour toggle: P_Rum_5_356.arrfbLysGruppe[1].fbLightCtrl.bDimUp
    Rectangle (127,252 71x22), "Dim Dwn", colour toggle: P_Rum_5_356.arrfbLysGruppe[1].fbLightCtrl.bDimDwn
    Ellipse (45,219 22x23), colour toggle: P_Rum_5_356.arrfbLysGruppe[1].fbLightCtrl.bAutoZone1
    Rectangle (78,219 122x22), "Lys Auto"
    Ellipse (45,54 22x23), colour toggle: P_Gang_5_356.arrfbLysGruppe[1].fbLightCtrl.bPIR
    Rectangle (77,54 122x22), "PIR status"
END_VISUALIZATION

// ---- POUs/Alle_Rum/Rum_Med_DALI_Pir/Rum_1_218/Visualization_5_356_2_1_1.TcVIS
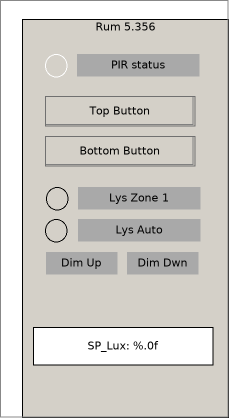
VISUALIZATION Visualization_5_356_2_1_1  // 229x418
    RoundedRectangle (22,19 207x399), "Rum 5.356"
    Rectangle (33,327 180x38), "SP_Lux: %.0f", text variable: P_Rum_5_356.arrfbLysGruppe[1].fbLightCtrl.fLuxZone1
    Button (45,96 150x30), "Top Button"
        tap P_Rum_5_356.bTopButtonZone1_Visu
    Button (45,136 150x30), "Bottom Button"
        tap P_Rum_5_356.bBottomButtonZone1_Visu
    Ellipse (46,187 22x23), colour toggle: P_Rum_5_356.arrfbLysGruppe[1].fbLightCtrl.bOnZone1
    Rectangle (78,187 122x22), "Lys Zone 1"
    Rectangle (46,252 71x22), "Dim Up", colour toggle: P_Rum_5_356.arrfbLysGruppe[1].fbLightCtrl.bDimUp
    Rectangle (127,252 71x22), "Dim Dwn", colour toggle: P_Rum_5_356.arrfbLysGruppe[1].fbLightCtrl.bDimDwn
    Ellipse (45,219 22x23), colour toggle: P_Rum_5_356.arrfbLysGruppe[1].fbLightCtrl.bAutoZone1
    Rectangle (78,219 122x22), "Lys Auto"
    Ellipse (45,54 22x23), colour toggle: P_Gang_5_356.arrfbLysGruppe[1].fbLightCtrl.bPIR
    Rectangle (77,54 122x22), "PIR status"
END_VISUALIZATION

// ---- POUs/Alle_Rum/Rum_Med_DALI_Pir/Rum_6_223/Visualization_5_356_2_1_1_6_1.TcVIS
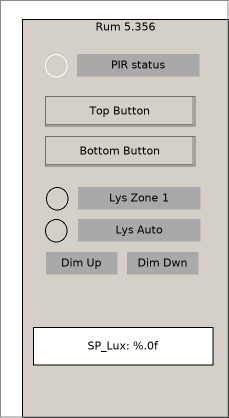
VISUALIZATION Visualization_5_356_2_1_1_6_1  // 229x418
    RoundedRectangle (22,19 207x399), "Rum 5.356"
    Rectangle (33,327 180x38), "SP_Lux: %.0f", text variable: P_Rum_5_356.arrfbLysGruppe[1].fbLightCtrl.fLuxZone1
    Button (45,96 150x30), "Top Button"
        tap P_Rum_5_356.bTopButtonZone1_Visu
    Button (45,136 150x30), "Bottom Button"
        tap P_Rum_5_356.bBottomButtonZone1_Visu
    Ellipse (46,187 22x23), colour toggle: P_Rum_5_356.arrfbLysGruppe[1].fbLightCtrl.bOnZone1
    Rectangle (78,187 122x22), "Lys Zone 1"
    Rectangle (46,252 71x22), "Dim Up", colour toggle: P_Rum_5_356.arrfbLysGruppe[1].fbLightCtrl.bDimUp
    Rectangle (127,252 71x22), "Dim Dwn", colour toggle: P_Rum_5_356.arrfbLysGruppe[1].fbLightCtrl.bDimDwn
    Ellipse (45,219 22x23), colour toggle: P_Rum_5_356.arrfbLysGruppe[1].fbLightCtrl.bAutoZone1
    Rectangle (78,219 122x22), "Lys Auto"
    Ellipse (45,54 22x23), colour toggle: P_Gang_5_356.arrfbLysGruppe[1].fbLightCtrl.bPIR
    Rectangle (77,54 122x22), "PIR status"
END_VISUALIZATION

// ---- POUs/Alle_Rum/Rum_Med_DALI_Pir/Rum_6_225/Visualization_5_356_2_1_1_6_1_10.TcVIS
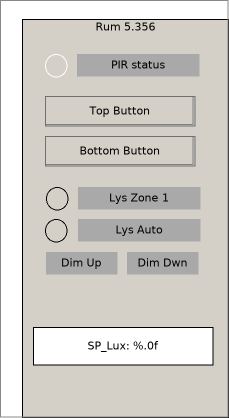
VISUALIZATION Visualization_5_356_2_1_1_6_1_10  // 229x418
    RoundedRectangle (22,19 207x399), "Rum 5.356"
    Rectangle (33,327 180x38), "SP_Lux: %.0f", text variable: P_Rum_5_356.arrfbLysGruppe[1].fbLightCtrl.fLuxZone1
    Button (45,96 150x30), "Top Button"
        tap P_Rum_5_356.bTopButtonZone1_Visu
    Button (45,136 150x30), "Bottom Button"
        tap P_Rum_5_356.bBottomButtonZone1_Visu
    Ellipse (46,187 22x23), colour toggle: P_Rum_5_356.arrfbLysGruppe[1].fbLightCtrl.bOnZone1
    Rectangle (78,187 122x22), "Lys Zone 1"
    Rectangle (46,252 71x22), "Dim Up", colour toggle: P_Rum_5_356.arrfbLysGruppe[1].fbLightCtrl.bDimUp
    Rectangle (127,252 71x22), "Dim Dwn", colour toggle: P_Rum_5_356.arrfbLysGruppe[1].fbLightCtrl.bDimDwn
    Ellipse (45,219 22x23), colour toggle: P_Rum_5_356.arrfbLysGruppe[1].fbLightCtrl.bAutoZone1
    Rectangle (78,219 122x22), "Lys Auto"
    Ellipse (45,54 22x23), colour toggle: P_Gang_5_356.arrfbLysGruppe[1].fbLightCtrl.bPIR
    Rectangle (77,54 122x22), "PIR status"
END_VISUALIZATION

// ---- POUs/Alle_Rum/Rum_Med_DALI_Pir/Rum_6_224/Visualization_5_356_2_1_1_6_1_1.TcVIS
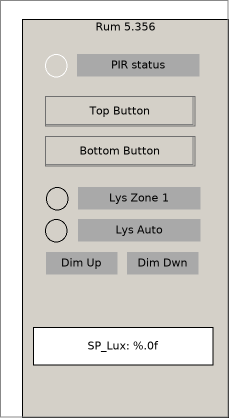
VISUALIZATION Visualization_5_356_2_1_1_6_1_1  // 229x418
    RoundedRectangle (22,19 207x399), "Rum 5.356"
    Rectangle (33,327 180x38), "SP_Lux: %.0f", text variable: P_Rum_5_356.arrfbLysGruppe[1].fbLightCtrl.fLuxZone1
    Button (45,96 150x30), "Top Button"
        tap P_Rum_5_356.bTopButtonZone1_Visu
    Button (45,136 150x30), "Bottom Button"
        tap P_Rum_5_356.bBottomButtonZone1_Visu
    Ellipse (46,187 22x23), colour toggle: P_Rum_5_356.arrfbLysGruppe[1].fbLightCtrl.bOnZone1
    Rectangle (78,187 122x22), "Lys Zone 1"
    Rectangle (46,252 71x22), "Dim Up", colour toggle: P_Rum_5_356.arrfbLysGruppe[1].fbLightCtrl.bDimUp
    Rectangle (127,252 71x22), "Dim Dwn", colour toggle: P_Rum_5_356.arrfbLysGruppe[1].fbLightCtrl.bDimDwn
    Ellipse (45,219 22x23), colour toggle: P_Rum_5_356.arrfbLysGruppe[1].fbLightCtrl.bAutoZone1
    Rectangle (78,219 122x22), "Lys Auto"
    Ellipse (45,54 22x23), colour toggle: P_Gang_5_356.arrfbLysGruppe[1].fbLightCtrl.bPIR
    Rectangle (77,54 122x22), "PIR status"
END_VISUALIZATION

// ---- POUs/Alle_Rum/Rum_Med_DALI_Pir/Rum_6_226A/Visualization_5_356_2_1_1_6_1_2.TcVIS
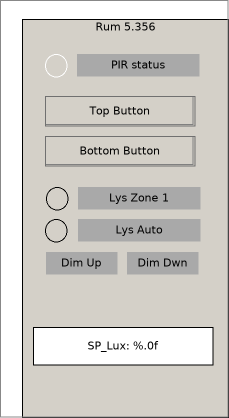
VISUALIZATION Visualization_5_356_2_1_1_6_1_2  // 229x418
    RoundedRectangle (22,19 207x399), "Rum 5.356"
    Rectangle (33,327 180x38), "SP_Lux: %.0f", text variable: P_Rum_5_356.arrfbLysGruppe[1].fbLightCtrl.fLuxZone1
    Button (45,96 150x30), "Top Button"
        tap P_Rum_5_356.bTopButtonZone1_Visu
    Button (45,136 150x30), "Bottom Button"
        tap P_Rum_5_356.bBottomButtonZone1_Visu
    Ellipse (46,187 22x23), colour toggle: P_Rum_5_356.arrfbLysGruppe[1].fbLightCtrl.bOnZone1
    Rectangle (78,187 122x22), "Lys Zone 1"
    Rectangle (46,252 71x22), "Dim Up", colour toggle: P_Rum_5_356.arrfbLysGruppe[1].fbLightCtrl.bDimUp
    Rectangle (127,252 71x22), "Dim Dwn", colour toggle: P_Rum_5_356.arrfbLysGruppe[1].fbLightCtrl.bDimDwn
    Ellipse (45,219 22x23), colour toggle: P_Rum_5_356.arrfbLysGruppe[1].fbLightCtrl.bAutoZone1
    Rectangle (78,219 122x22), "Lys Auto"
    Ellipse (45,54 22x23), colour toggle: P_Gang_5_356.arrfbLysGruppe[1].fbLightCtrl.bPIR
    Rectangle (77,54 122x22), "PIR status"
END_VISUALIZATION

// ---- POUs/Alle_Rum/Rum_Med_DALI_Pir/Rum_6_227/Visualization_5_356_2_1_1_6_1_3.TcVIS
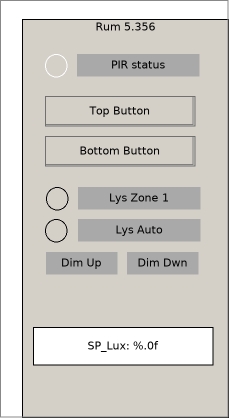
VISUALIZATION Visualization_5_356_2_1_1_6_1_3  // 229x418
    RoundedRectangle (22,19 207x399), "Rum 5.356"
    Rectangle (33,327 180x38), "SP_Lux: %.0f", text variable: P_Rum_5_356.arrfbLysGruppe[1].fbLightCtrl.fLuxZone1
    Button (45,96 150x30), "Top Button"
        tap P_Rum_5_356.bTopButtonZone1_Visu
    Button (45,136 150x30), "Bottom Button"
        tap P_Rum_5_356.bBottomButtonZone1_Visu
    Ellipse (46,187 22x23), colour toggle: P_Rum_5_356.arrfbLysGruppe[1].fbLightCtrl.bOnZone1
    Rectangle (78,187 122x22), "Lys Zone 1"
    Rectangle (46,252 71x22), "Dim Up", colour toggle: P_Rum_5_356.arrfbLysGruppe[1].fbLightCtrl.bDimUp
    Rectangle (127,252 71x22), "Dim Dwn", colour toggle: P_Rum_5_356.arrfbLysGruppe[1].fbLightCtrl.bDimDwn
    Ellipse (45,219 22x23), colour toggle: P_Rum_5_356.arrfbLysGruppe[1].fbLightCtrl.bAutoZone1
    Rectangle (78,219 122x22), "Lys Auto"
    Ellipse (45,54 22x23), colour toggle: P_Gang_5_356.arrfbLysGruppe[1].fbLightCtrl.bPIR
    Rectangle (77,54 122x22), "PIR status"
END_VISUALIZATION

// ---- POUs/Alle_Rum/Rum_Med_DALI_Pir/Rum_6_228/Visualization_5_356_2_1_1_6_1_4.TcVIS
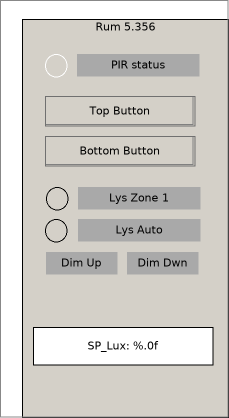
VISUALIZATION Visualization_5_356_2_1_1_6_1_4  // 229x418
    RoundedRectangle (22,19 207x399), "Rum 5.356"
    Rectangle (33,327 180x38), "SP_Lux: %.0f", text variable: P_Rum_5_356.arrfbLysGruppe[1].fbLightCtrl.fLuxZone1
    Button (45,96 150x30), "Top Button"
        tap P_Rum_5_356.bTopButtonZone1_Visu
    Button (45,136 150x30), "Bottom Button"
        tap P_Rum_5_356.bBottomButtonZone1_Visu
    Ellipse (46,187 22x23), colour toggle: P_Rum_5_356.arrfbLysGruppe[1].fbLightCtrl.bOnZone1
    Rectangle (78,187 122x22), "Lys Zone 1"
    Rectangle (46,252 71x22), "Dim Up", colour toggle: P_Rum_5_356.arrfbLysGruppe[1].fbLightCtrl.bDimUp
    Rectangle (127,252 71x22), "Dim Dwn", colour toggle: P_Rum_5_356.arrfbLysGruppe[1].fbLightCtrl.bDimDwn
    Ellipse (45,219 22x23), colour toggle: P_Rum_5_356.arrfbLysGruppe[1].fbLightCtrl.bAutoZone1
    Rectangle (78,219 122x22), "Lys Auto"
    Ellipse (45,54 22x23), colour toggle: P_Gang_5_356.arrfbLysGruppe[1].fbLightCtrl.bPIR
    Rectangle (77,54 122x22), "PIR status"
END_VISUALIZATION

// ---- POUs/Alle_Rum/Rum_Med_DALI_Pir/Rum_6_229/Visualization_5_356_2_1_1_6_1_5.TcVIS
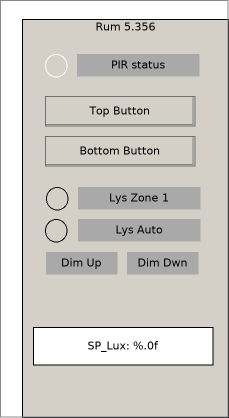
VISUALIZATION Visualization_5_356_2_1_1_6_1_5  // 229x418
    RoundedRectangle (22,19 207x399), "Rum 5.356"
    Rectangle (33,327 180x38), "SP_Lux: %.0f", text variable: P_Rum_5_356.arrfbLysGruppe[1].fbLightCtrl.fLuxZone1
    Button (45,96 150x30), "Top Button"
        tap P_Rum_5_356.bTopButtonZone1_Visu
    Button (45,136 150x30), "Bottom Button"
        tap P_Rum_5_356.bBottomButtonZone1_Visu
    Ellipse (46,187 22x23), colour toggle: P_Rum_5_356.arrfbLysGruppe[1].fbLightCtrl.bOnZone1
    Rectangle (78,187 122x22), "Lys Zone 1"
    Rectangle (46,252 71x22), "Dim Up", colour toggle: P_Rum_5_356.arrfbLysGruppe[1].fbLightCtrl.bDimUp
    Rectangle (127,252 71x22), "Dim Dwn", colour toggle: P_Rum_5_356.arrfbLysGruppe[1].fbLightCtrl.bDimDwn
    Ellipse (45,219 22x23), colour toggle: P_Rum_5_356.arrfbLysGruppe[1].fbLightCtrl.bAutoZone1
    Rectangle (78,219 122x22), "Lys Auto"
    Ellipse (45,54 22x23), colour toggle: P_Gang_5_356.arrfbLysGruppe[1].fbLightCtrl.bPIR
    Rectangle (77,54 122x22), "PIR status"
END_VISUALIZATION

// ---- POUs/Alle_Rum/Rum_Med_DALI_Pir/Rum_6_230/Visualization_5_356_2_1_1_6_1_6.TcVIS
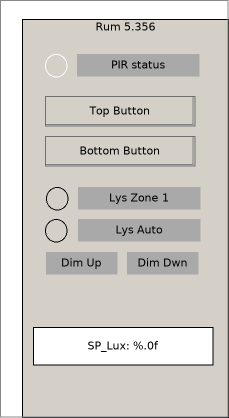
VISUALIZATION Visualization_5_356_2_1_1_6_1_6  // 229x418
    RoundedRectangle (22,19 207x399), "Rum 5.356"
    Rectangle (33,327 180x38), "SP_Lux: %.0f", text variable: P_Rum_5_356.arrfbLysGruppe[1].fbLightCtrl.fLuxZone1
    Button (45,96 150x30), "Top Button"
        tap P_Rum_5_356.bTopButtonZone1_Visu
    Button (45,136 150x30), "Bottom Button"
        tap P_Rum_5_356.bBottomButtonZone1_Visu
    Ellipse (46,187 22x23), colour toggle: P_Rum_5_356.arrfbLysGruppe[1].fbLightCtrl.bOnZone1
    Rectangle (78,187 122x22), "Lys Zone 1"
    Rectangle (46,252 71x22), "Dim Up", colour toggle: P_Rum_5_356.arrfbLysGruppe[1].fbLightCtrl.bDimUp
    Rectangle (127,252 71x22), "Dim Dwn", colour toggle: P_Rum_5_356.arrfbLysGruppe[1].fbLightCtrl.bDimDwn
    Ellipse (45,219 22x23), colour toggle: P_Rum_5_356.arrfbLysGruppe[1].fbLightCtrl.bAutoZone1
    Rectangle (78,219 122x22), "Lys Auto"
    Ellipse (45,54 22x23), colour toggle: P_Gang_5_356.arrfbLysGruppe[1].fbLightCtrl.bPIR
    Rectangle (77,54 122x22), "PIR status"
END_VISUALIZATION

// ---- POUs/Alle_Rum/Rum_Med_DALI_Pir/Rum_6_231/Visualization_5_356_2_1_1_6_1_7.TcVIS
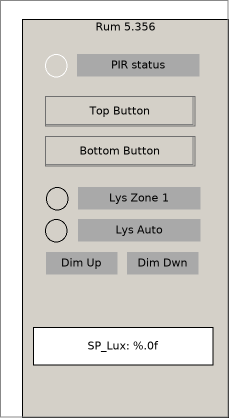
VISUALIZATION Visualization_5_356_2_1_1_6_1_7  // 229x418
    RoundedRectangle (22,19 207x399), "Rum 5.356"
    Rectangle (33,327 180x38), "SP_Lux: %.0f", text variable: P_Rum_5_356.arrfbLysGruppe[1].fbLightCtrl.fLuxZone1
    Button (45,96 150x30), "Top Button"
        tap P_Rum_5_356.bTopButtonZone1_Visu
    Button (45,136 150x30), "Bottom Button"
        tap P_Rum_5_356.bBottomButtonZone1_Visu
    Ellipse (46,187 22x23), colour toggle: P_Rum_5_356.arrfbLysGruppe[1].fbLightCtrl.bOnZone1
    Rectangle (78,187 122x22), "Lys Zone 1"
    Rectangle (46,252 71x22), "Dim Up", colour toggle: P_Rum_5_356.arrfbLysGruppe[1].fbLightCtrl.bDimUp
    Rectangle (127,252 71x22), "Dim Dwn", colour toggle: P_Rum_5_356.arrfbLysGruppe[1].fbLightCtrl.bDimDwn
    Ellipse (45,219 22x23), colour toggle: P_Rum_5_356.arrfbLysGruppe[1].fbLightCtrl.bAutoZone1
    Rectangle (78,219 122x22), "Lys Auto"
    Ellipse (45,54 22x23), colour toggle: P_Gang_5_356.arrfbLysGruppe[1].fbLightCtrl.bPIR
    Rectangle (77,54 122x22), "PIR status"
END_VISUALIZATION

// ---- POUs/Alle_Rum/Rum_Med_DALI_Pir/Rum_6_233/Visualization_5_356_2_1_1_6_1_8.TcVIS
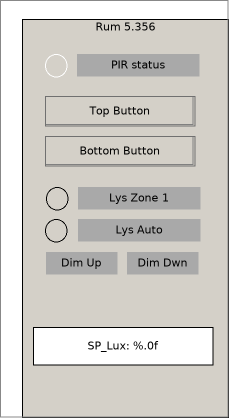
VISUALIZATION Visualization_5_356_2_1_1_6_1_8  // 229x418
    RoundedRectangle (22,19 207x399), "Rum 5.356"
    Rectangle (33,327 180x38), "SP_Lux: %.0f", text variable: P_Rum_5_356.arrfbLysGruppe[1].fbLightCtrl.fLuxZone1
    Button (45,96 150x30), "Top Button"
        tap P_Rum_5_356.bTopButtonZone1_Visu
    Button (45,136 150x30), "Bottom Button"
        tap P_Rum_5_356.bBottomButtonZone1_Visu
    Ellipse (46,187 22x23), colour toggle: P_Rum_5_356.arrfbLysGruppe[1].fbLightCtrl.bOnZone1
    Rectangle (78,187 122x22), "Lys Zone 1"
    Rectangle (46,252 71x22), "Dim Up", colour toggle: P_Rum_5_356.arrfbLysGruppe[1].fbLightCtrl.bDimUp
    Rectangle (127,252 71x22), "Dim Dwn", colour toggle: P_Rum_5_356.arrfbLysGruppe[1].fbLightCtrl.bDimDwn
    Ellipse (45,219 22x23), colour toggle: P_Rum_5_356.arrfbLysGruppe[1].fbLightCtrl.bAutoZone1
    Rectangle (78,219 122x22), "Lys Auto"
    Ellipse (45,54 22x23), colour toggle: P_Gang_5_356.arrfbLysGruppe[1].fbLightCtrl.bPIR
    Rectangle (77,54 122x22), "PIR status"
END_VISUALIZATION

// ---- POUs/DALI/DALI_Setup/VISUs/TextLists/CommandOnTerminalEvent.TcTLO
TEXTLIST CommandOnTerminalEvent
  0 = 'Do Nothing'
  1 = 'Off'
  2 = 'RecallMaxLevel'
  3 = 'RecallMinLevel'
  4 = 'GoToScene0'
  5 = 'GoToScene1'
  6 = 'GoToScene2'
  7 = 'GoToScene3'
  8 = 'GoToScene4'
  9 = 'GoToScene5'
  10 = 'GoToScene6'
  11 = 'GoToScene7'
  12 = 'GoToScene8'
  13 = 'GoToScene9'
  14 = 'GoToScene10'
  15 = 'GoToScene11'
  16 = 'GoToScene12'
  17 = 'GoToScene13'
  18 = 'GoToScene14'
  19 = 'GoToScene15'
   = ''
END_TEXTLIST

// ---- POUs/DALI/DALI_Setup/VISUs/TextLists/EventScheme.TcTLO
TEXTLIST EventScheme
  0 = '0 - Instance type and number'
  1 = '1 - Short address and instance type'
  2 = '2 - Short address and instance number'
  3 = '3 - Device group and instance type'
  4 = '4 - Instance group and instance type'
   = ''
END_TEXTLIST

// ---- POUs/DALI/DALI_Setup/VISUs/TextLists/ExtendedFadeTime.TcTLO
TEXTLIST ExtendedFadeTime
  0 = 'No Fade'
  1 = '1 * 100 ms = 100 ms'
  2 = '2 * 100 ms = 200 ms'
  3 = '3 * 100 ms = 300 ms'
  4 = '4 * 100 ms = 400 ms'
  5 = '5 * 100 ms = 500 ms'
  6 = '6 * 100 ms = 600 ms'
  7 = '7 * 100 ms = 700 ms'
  8 = '8 * 100 ms = 800 ms'
  9 = '9 * 100 ms = 900 ms'
  10 = '10 * 100 ms = 1000 ms'
  11 = '11 * 100 ms = 1100 ms'
  12 = '12 * 100 ms = 1200 ms'
  13 = '13 * 100 ms = 1300 ms'
  14 = '14 * 100 ms = 1400 ms'
  15 = '15 * 100 ms = 1500 ms'
  16 = '16 * 100 ms = 1600 ms'
  17 = '1 * 1 s = 1 s'
  18 = '2 * 1 s = 2 s'
  19 = '3 * 1 s = 3 s'
  20 = '4 * 1 s = 4 s'
  21 = '5 * 1 s = 5 s'
  22 = '6 * 1 s = 6 s'
  23 = '7 * 1 s = 7 s'
  24 = '8 * 1 s = 8 s'
  25 = '9 * 1 s = 9 s'
  26 = '10 * 1 s = 10 s'
  27 = '11 * 1 s = 11 s'
  28 = '12 * 1 s = 12 s'
  29 = '13 * 1 s = 13 s'
  30 = '14 * 1 s = 14 s'
  31 = '15 * 1 s = 15 s'
  32 = '16 * 1 s = 16 s'
  33 = '1 * 10 s = 10 s'
  34 = '2 * 10 s = 20 s'
  35 = '3 * 10 s = 30 s'
  36 = '4 * 10 s = 40 s'
  37 = '5 * 10 s = 50 s'
  38 = '6 * 10 s = 60 s'
  39 = '7 * 10 s = 70 s'
  40 = '8 * 10 s = 80 s'
  41 = '9 * 10 s = 90 s'
  42 = '10 * 10 s = 100 s'
  43 = '11 * 10 s = 110 s'
  44 = '12 * 10 s = 120 s'
  45 = '13 * 10 s = 130 s'
  46 = '14 * 10 s = 140 s'
  47 = '15 * 10 s = 150 s'
  48 = '16 * 10 s = 160 s'
  49 = '1 * 1 min = 1 min'
  50 = '2 * 1 min = 2 min'
  51 = '3 * 1 min = 3 min'
  52 = '4 * 1 min = 4 min'
  53 = '5 * 1 min = 5 min'
  54 = '6 * 1 min = 6 min'
  55 = '7 * 1 min = 7 min'
  56 = '8 * 1 min = 8 min'
  57 = '9 * 1 min = 9 min'
  58 = '10 * 1 min = 10 min'
  59 = '11 * 1 min = 11 min'
  60 = '12 * 1 min = 12 min'
  61 = '13 * 1 min = 13 min'
  62 = '14 * 1 min = 14 min'
  63 = '15 * 1 min = 15 min'
  64 = '16 * 1 min = 16 min'
  255 = 'Unknown'
   = ''
END_TEXTLIST

// ---- POUs/DALI/DALI_Setup/VISUs/Visu_DALICommissioning.TcVIS
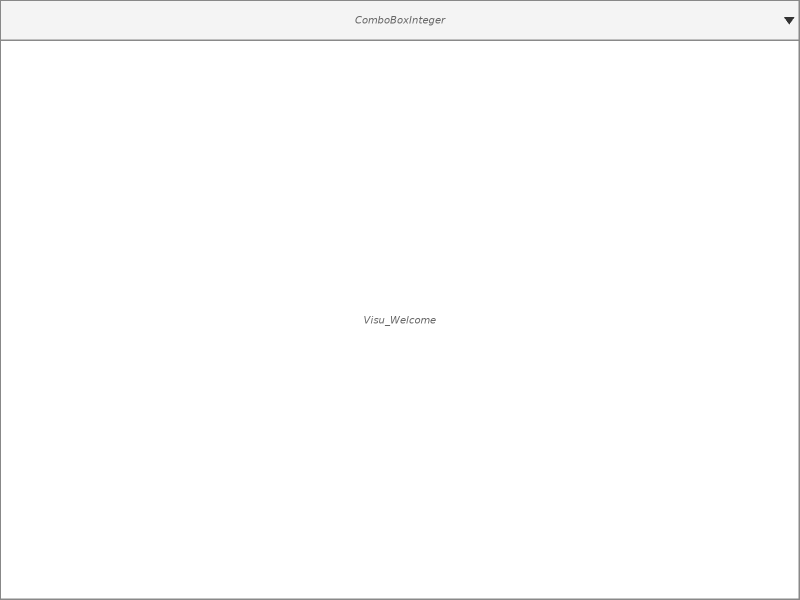
VISUALIZATION Visu_DALICommissioning  // 800x600
    ComboBoxInteger (0,0 800x40), variable: DALI_Commissioning.nSelectedDialog, input disabled if: DALI_Commissioning.bDisableComboBox, text list: 'TextList_Dialogs'
    Frame (0,40 800x560), frame switch variable: DALI_Commissioning.nSelectedDialog
        shows Visu_Welcome()
        shows Visu_Part102Commands()
        shows Visu_Part102Addressing()
        shows Visu_Part102Parameters()
        shows Visu_Part102Groups()
        shows Visu_Part102Scenes()
        shows Visu_Part102MemoryBank()
        shows Visu_Part102SetFading()
        shows Visu_Part202()
        shows Visu_Part205()
        shows Visu_Part207()
        shows Visu_Part208Switching()
        shows Visu_Part103Addressing()
        shows Visu_Part103Parameters()
        shows Visu_Part103Identify()
        shows Visu_Part301PushButton()
        shows Visu_Part302AbsoluteInputDevice()
        shows Visu_Part303OccupancySensor()
        shows Visu_Part304LightSensor()
        shows Visu_Part300GenericDevice()
        shows Visu_Part103MemoryBank()
        shows Visu_KL6821Configuration()
END_VISUALIZATION

// ---- POUs/DALI/DALI_Setup/VISUs/Visu_DALICommissioning/Visu_Part102Addressing.TcVIS
